FUNCTION_BLOCK SS3_ifb_Camera (* Basic FB with empty ECC *)
  (* Standard: 61499-2 *)
  (* Version 1.0, 2021-08-03, AK121668 *)
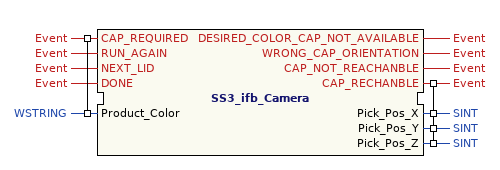
  EVENT_INPUT
    CAP_REQUIRED WITH Product_Color;
    RUN_AGAIN;
    NEXT_LID;
    DONE;
  END_EVENT
  EVENT_OUTPUT
    DESIRED_COLOR_CAP_NOT_AVAILABLE;
    WRONG_CAP_ORIENTATION;
    CAP_NOT_REACHANBLE;
    CAP_RECHANBLE WITH Pick_Pos_X, Pick_Pos_Y, Pick_Pos_Z;
  END_EVENT
  VAR_INPUT
    Product_Color : WSTRING;
  END_VAR
  VAR_OUTPUT
    Pick_Pos_X : SINT;
    Pick_Pos_Y : SINT;
    Pick_Pos_Z : SINT;
  END_VAR
  VAR
    ifg_desiredCapNotAvailable : BOOL;
    ifg_wrong_orientation : BOOL;
    ifg_cap_not_reachable : BOOL;
    ifg_cap_reachable : BOOL;
  END_VAR
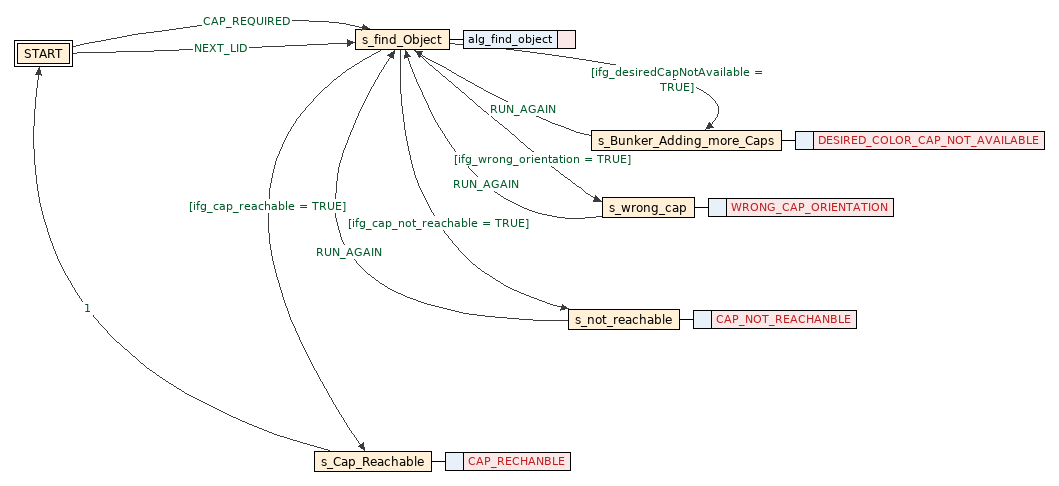
  EC_STATES
    START; (* Initial State *)
    s_find_Object : alg_find_object;
    s_Bunker_Adding_more_Caps : -> DESIRED_COLOR_CAP_NOT_AVAILABLE;
    s_Cap_Reachable : -> CAP_RECHANBLE;
    s_wrong_cap : -> WRONG_CAP_ORIENTATION;
    s_not_reachable : -> CAP_NOT_REACHANBLE;
  END_STATES
  EC_TRANSITIONS
    START TO s_find_Object := CAP_REQUIRED;
    s_find_Object TO s_Bunker_Adding_more_Caps := [ifg_desiredCapNotAvailable = TRUE];
    s_find_Object TO s_wrong_cap := [ifg_wrong_orientation = TRUE];
    s_find_Object TO s_not_reachable := [ifg_cap_not_reachable = TRUE];
    s_Bunker_Adding_more_Caps TO s_find_Object := RUN_AGAIN;
    s_wrong_cap TO s_find_Object := RUN_AGAIN;
    s_not_reachable TO s_find_Object := RUN_AGAIN;
    s_find_Object TO s_Cap_Reachable := [ifg_cap_reachable = TRUE];
    s_Cap_Reachable TO START := 1;
    START TO s_find_Object := NEXT_LID;
  END_TRANSITIONS
  ALGORITHM alg_find_object IN ST:
//
Pick_Pos_X := 100;
Pick_Pos_Y := 50;
Pick_Pos_Z := 5;
  END_ALGORITHM
END_FUNCTION_BLOCK
